// Copyright (c) 2024 Loupe (https://loupe.team), provided under the MIT License.
TYPE AbbLinkinAuth_Typ :
STRUCT
	numAttempts : UINT;
	wwwAuthContent : ABBLINKIN_STRING_EX_LEN;
	digest : AbbLinkinAuthDigest_Typ;
	httpSessionCookie : STRING;
	ABBCXCookie : STRING;
END_STRUCT
END_TYPE

(* stored: Version 1.1.0.1, ProductVersion 3.1.4024.12
   DUT AbbLinkinAuth_Typ: Id {3b3e7797-3422-4ef6-95c4-998015db4fcc} *)
